{attribute 'qualified_only'}
{attribute 'strict'}
TYPE eTcoAimTtiPowerSupplyTests :
(
    Restore := 1,
    CleanUp,
    Message,
    PowerDisable,
    PowerEnable,
    Reset,
    MoveRelativePositiveWithDisabledPositiveDirection,
    MoveRelativePositiveWithEnabledPositiveDirection,
    MoveRelativeNegativeWithDisabledNegativeDirection,
    MoveRelativeNegativeWithEnabledNegativeDirection,
    HommingDirect,
    MoveVelocityPositiveWithDisabledPositiveDirection,
    MoveVelocityPositiveWithEnabledPositiveDirection,
    Stop,
    MoveVelocityNegativeWithDisabledNegativeDirection,
    MoveVelocityNegativeWithEnabledNegativeDirection,
	MoveAbsoluteDisabled,
	MoveAbsoluteDisabledPositiveDirection,
	MoveAbsoluteEnabledPositiveDirection,
	MoveAbsoluteDisabledNegativeDirection,
	MoveAbsoluteEnabledNegativeDirection,
	
    Last
);
END_TYPE

(* stored: Version 1.1.0.1, ProductVersion 3.1.4024.12
   DUT eTcoAimTtiPowerSupplyTests: Id {f2a00a44-6906-068c-16e5-c34f2e71ab27} *)
